// TIA Portal V19 export
FUNCTION "INPUT MAPING" : Void   // FC1, LAD
{ S7_Optimized_Access := 'TRUE' }
// stored: SetENOAutomatically false
BEGIN

REGION Network 1: "CPU RUN"
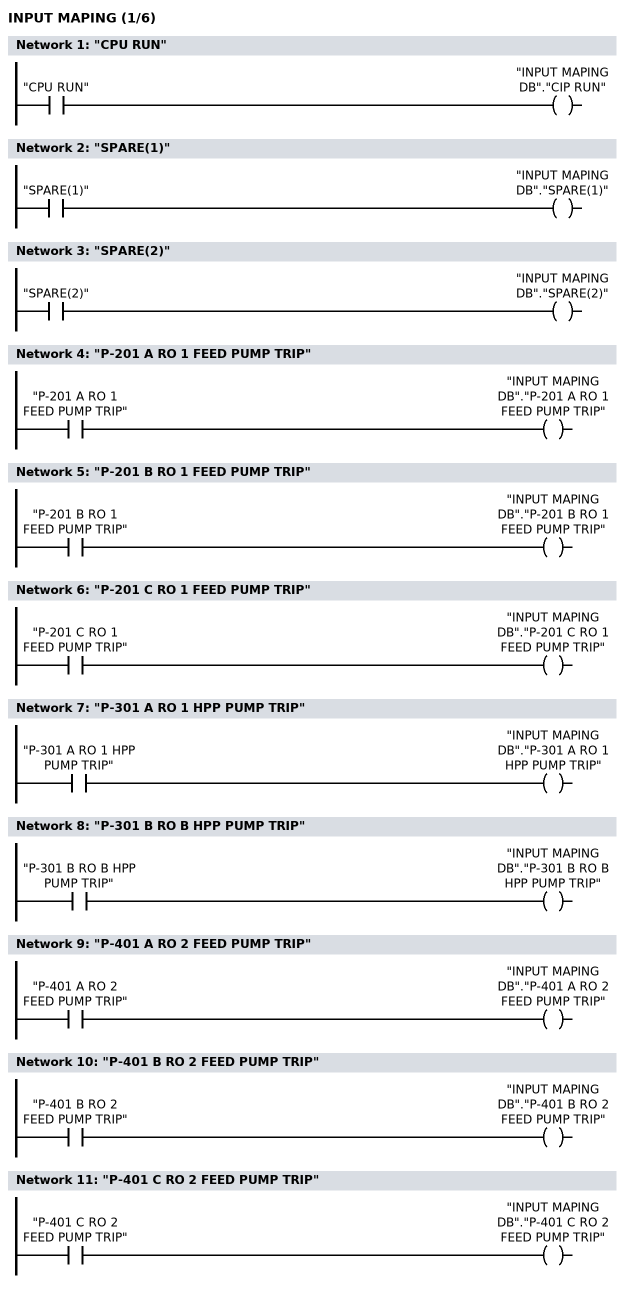
   RUNG wire#powerrail
      Contact( "CPU RUN" )
      Coil( "INPUT MAPING DB"."CIP RUN" )
   END_RUNG
   // the same network as SCL:
   "INPUT MAPING DB"."CIP RUN" := "CPU RUN";
END_REGION

REGION Network 2: "SPARE(1)"
   RUNG wire#powerrail
      Contact( "SPARE(1)" )
      Coil( "INPUT MAPING DB"."SPARE(1)" )
   END_RUNG
   // the same network as SCL:
   "INPUT MAPING DB"."SPARE(1)" := "SPARE(1)";
END_REGION

REGION Network 3: "SPARE(2)"
   RUNG wire#powerrail
      Contact( "SPARE(2)" )
      Coil( "INPUT MAPING DB"."SPARE(2)" )
   END_RUNG
   // the same network as SCL:
   "INPUT MAPING DB"."SPARE(2)" := "SPARE(2)";
END_REGION

REGION Network 4: "P-201 A RO 1 FEED PUMP TRIP"
   RUNG wire#powerrail
      Contact( "P-201 A RO 1 FEED PUMP TRIP" )
      Coil( "INPUT MAPING DB"."P-201 A RO 1 FEED PUMP TRIP" )
   END_RUNG
   // the same network as SCL:
   "INPUT MAPING DB"."P-201 A RO 1 FEED PUMP TRIP" := "P-201 A RO 1 FEED PUMP TRIP";
END_REGION

REGION Network 5: "P-201 B RO 1 FEED PUMP TRIP"
   RUNG wire#powerrail
      Contact( "P-201 B RO 1 FEED PUMP TRIP" )
      Coil( "INPUT MAPING DB"."P-201 B RO 1 FEED PUMP TRIP" )
   END_RUNG
   // the same network as SCL:
   "INPUT MAPING DB"."P-201 B RO 1 FEED PUMP TRIP" := "P-201 B RO 1 FEED PUMP TRIP";
END_REGION

REGION Network 6: "P-201 C RO 1 FEED PUMP TRIP"
   RUNG wire#powerrail
      Contact( "P-201 C RO 1 FEED PUMP TRIP" )
      Coil( "INPUT MAPING DB"."P-201 C RO 1 FEED PUMP TRIP" )
   END_RUNG
   // the same network as SCL:
   "INPUT MAPING DB"."P-201 C RO 1 FEED PUMP TRIP" := "P-201 C RO 1 FEED PUMP TRIP";
END_REGION

REGION Network 7: "P-301 A RO 1 HPP PUMP TRIP"
   RUNG wire#powerrail
      Contact( "P-301 A RO 1 HPP PUMP TRIP" )
      Coil( "INPUT MAPING DB"."P-301 A RO 1 HPP PUMP TRIP" )
   END_RUNG
   // the same network as SCL:
   "INPUT MAPING DB"."P-301 A RO 1 HPP PUMP TRIP" := "P-301 A RO 1 HPP PUMP TRIP";
END_REGION

REGION Network 8: "P-301 B RO B HPP PUMP TRIP"
   RUNG wire#powerrail
      Contact( "P-301 B RO B HPP PUMP TRIP" )
      Coil( "INPUT MAPING DB"."P-301 B RO B HPP PUMP TRIP" )
   END_RUNG
   // the same network as SCL:
   "INPUT MAPING DB"."P-301 B RO B HPP PUMP TRIP" := "P-301 B RO B HPP PUMP TRIP";
END_REGION

REGION Network 9: "P-401 A RO 2 FEED PUMP TRIP"
   RUNG wire#powerrail
      Contact( "P-401 A RO 2 FEED PUMP TRIP" )
      Coil( "INPUT MAPING DB"."P-401 A RO 2 FEED PUMP TRIP" )
   END_RUNG
   // the same network as SCL:
   "INPUT MAPING DB"."P-401 A RO 2 FEED PUMP TRIP" := "P-401 A RO 2 FEED PUMP TRIP";
END_REGION

REGION Network 10: "P-401 B RO 2 FEED PUMP TRIP"
   RUNG wire#powerrail
      Contact( "P-401 B RO 2 FEED PUMP TRIP" )
      Coil( "INPUT MAPING DB"."P-401 B RO 2 FEED PUMP TRIP" )
   END_RUNG
   // the same network as SCL:
   "INPUT MAPING DB"."P-401 B RO 2 FEED PUMP TRIP" := "P-401 B RO 2 FEED PUMP TRIP";
END_REGION

REGION Network 11: "P-401 C RO 2 FEED PUMP TRIP"
   RUNG wire#powerrail
      Contact( "P-401 C RO 2 FEED PUMP TRIP" )
      Coil( "INPUT MAPING DB"."P-401 C RO 2 FEED PUMP TRIP" )
   END_RUNG
   // the same network as SCL:
   "INPUT MAPING DB"."P-401 C RO 2 FEED PUMP TRIP" := "P-401 C RO 2 FEED PUMP TRIP";
END_REGION

REGION Network 12: "P 401 A RO 2 HPP PUMP TRIP"
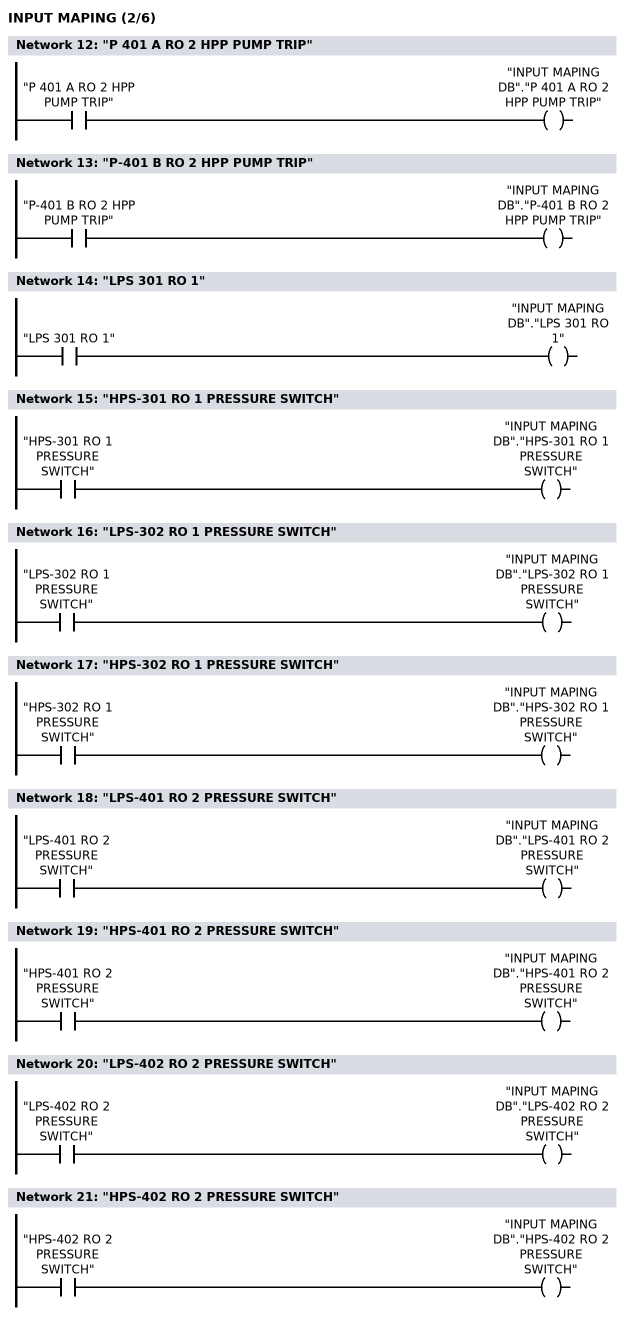
   RUNG wire#powerrail
      Contact( "P 401 A RO 2 HPP PUMP TRIP" )
      Coil( "INPUT MAPING DB"."P 401 A RO 2 HPP PUMP TRIP" )
   END_RUNG
   // the same network as SCL:
   "INPUT MAPING DB"."P 401 A RO 2 HPP PUMP TRIP" := "P 401 A RO 2 HPP PUMP TRIP";
END_REGION

REGION Network 13: "P-401 B RO 2 HPP PUMP TRIP"
   RUNG wire#powerrail
      Contact( "P-401 B RO 2 HPP PUMP TRIP" )
      Coil( "INPUT MAPING DB"."P-401 B RO 2 HPP PUMP TRIP" )
   END_RUNG
   // the same network as SCL:
   "INPUT MAPING DB"."P-401 B RO 2 HPP PUMP TRIP" := "P-401 B RO 2 HPP PUMP TRIP";
END_REGION

REGION Network 14: "LPS 301 RO 1"
   RUNG wire#powerrail
      Contact( "LPS 301 RO 1" )
      Coil( "INPUT MAPING DB"."LPS 301 RO 1" )
   END_RUNG
   // the same network as SCL:
   "INPUT MAPING DB"."LPS 301 RO 1" := "LPS 301 RO 1";
END_REGION

REGION Network 15: "HPS-301 RO 1 PRESSURE SWITCH"
   RUNG wire#powerrail
      Contact( "HPS-301 RO 1 PRESSURE SWITCH" )
      Coil( "INPUT MAPING DB"."HPS-301 RO 1 PRESSURE SWITCH" )
   END_RUNG
   // the same network as SCL:
   "INPUT MAPING DB"."HPS-301 RO 1 PRESSURE SWITCH" := "HPS-301 RO 1 PRESSURE SWITCH";
END_REGION

REGION Network 16: "LPS-302 RO 1 PRESSURE SWITCH"
   RUNG wire#powerrail
      Contact( "LPS-302 RO 1 PRESSURE SWITCH" )
      Coil( "INPUT MAPING DB"."LPS-302 RO 1 PRESSURE SWITCH" )
   END_RUNG
   // the same network as SCL:
   "INPUT MAPING DB"."LPS-302 RO 1 PRESSURE SWITCH" := "LPS-302 RO 1 PRESSURE SWITCH";
END_REGION

REGION Network 17: "HPS-302 RO 1 PRESSURE SWITCH"
   RUNG wire#powerrail
      Contact( "HPS-302 RO 1 PRESSURE SWITCH" )
      Coil( "INPUT MAPING DB"."HPS-302 RO 1 PRESSURE SWITCH" )
   END_RUNG
   // the same network as SCL:
   "INPUT MAPING DB"."HPS-302 RO 1 PRESSURE SWITCH" := "HPS-302 RO 1 PRESSURE SWITCH";
END_REGION

REGION Network 18: "LPS-401 RO 2 PRESSURE SWITCH"
   RUNG wire#powerrail
      Contact( "LPS-401 RO 2 PRESSURE SWITCH" )
      Coil( "INPUT MAPING DB"."LPS-401 RO 2 PRESSURE SWITCH" )
   END_RUNG
   // the same network as SCL:
   "INPUT MAPING DB"."LPS-401 RO 2 PRESSURE SWITCH" := "LPS-401 RO 2 PRESSURE SWITCH";
END_REGION

REGION Network 19: "HPS-401 RO 2 PRESSURE SWITCH"
   RUNG wire#powerrail
      Contact( "HPS-401 RO 2 PRESSURE SWITCH" )
      Coil( "INPUT MAPING DB"."HPS-401 RO 2 PRESSURE SWITCH" )
   END_RUNG
   // the same network as SCL:
   "INPUT MAPING DB"."HPS-401 RO 2 PRESSURE SWITCH" := "HPS-401 RO 2 PRESSURE SWITCH";
END_REGION

REGION Network 20: "LPS-402 RO 2 PRESSURE SWITCH"
   RUNG wire#powerrail
      Contact( "LPS-402 RO 2 PRESSURE SWITCH" )
      Coil( "INPUT MAPING DB"."LPS-402 RO 2 PRESSURE SWITCH" )
   END_RUNG
   // the same network as SCL:
   "INPUT MAPING DB"."LPS-402 RO 2 PRESSURE SWITCH" := "LPS-402 RO 2 PRESSURE SWITCH";
END_REGION

REGION Network 21: "HPS-402 RO 2 PRESSURE SWITCH"
   RUNG wire#powerrail
      Contact( "HPS-402 RO 2 PRESSURE SWITCH" )
      Coil( "INPUT MAPING DB"."HPS-402 RO 2 PRESSURE SWITCH" )
   END_RUNG
   // the same network as SCL:
   "INPUT MAPING DB"."HPS-402 RO 2 PRESSURE SWITCH" := "HPS-402 RO 2 PRESSURE SWITCH";
END_REGION

REGION Network 22: "DP-703 RO 1 DOSER LEVEL SWITCH"
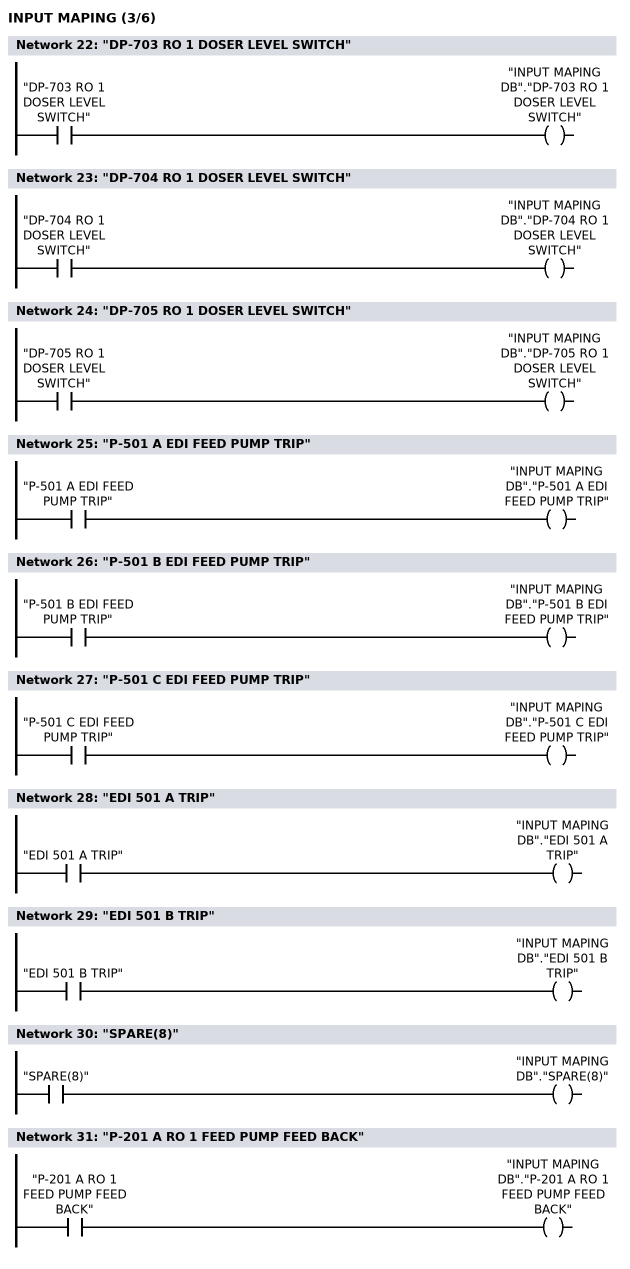
   RUNG wire#powerrail
      Contact( "DP-703 RO 1 DOSER LEVEL SWITCH" )
      Coil( "INPUT MAPING DB"."DP-703 RO 1 DOSER LEVEL SWITCH" )
   END_RUNG
   // the same network as SCL:
   "INPUT MAPING DB"."DP-703 RO 1 DOSER LEVEL SWITCH" := "DP-703 RO 1 DOSER LEVEL SWITCH";
END_REGION

REGION Network 23: "DP-704 RO 1 DOSER LEVEL SWITCH"
   RUNG wire#powerrail
      Contact( "DP-704 RO 1 DOSER LEVEL SWITCH" )
      Coil( "INPUT MAPING DB"."DP-704 RO 1 DOSER LEVEL SWITCH" )
   END_RUNG
   // the same network as SCL:
   "INPUT MAPING DB"."DP-704 RO 1 DOSER LEVEL SWITCH" := "DP-704 RO 1 DOSER LEVEL SWITCH";
END_REGION

REGION Network 24: "DP-705 RO 1 DOSER LEVEL SWITCH"
   RUNG wire#powerrail
      Contact( "DP-705 RO 1 DOSER LEVEL SWITCH" )
      Coil( "INPUT MAPING DB"."DP-705 RO 1 DOSER LEVEL SWITCH" )
   END_RUNG
   // the same network as SCL:
   "INPUT MAPING DB"."DP-705 RO 1 DOSER LEVEL SWITCH" := "DP-705 RO 1 DOSER LEVEL SWITCH";
END_REGION

REGION Network 25: "P-501 A EDI FEED PUMP TRIP"
   RUNG wire#powerrail
      Contact( "P-501 A EDI FEED PUMP TRIP" )
      Coil( "INPUT MAPING DB"."P-501 A EDI FEED PUMP TRIP" )
   END_RUNG
   // the same network as SCL:
   "INPUT MAPING DB"."P-501 A EDI FEED PUMP TRIP" := "P-501 A EDI FEED PUMP TRIP";
END_REGION

REGION Network 26: "P-501 B EDI FEED PUMP TRIP"
   RUNG wire#powerrail
      Contact( "P-501 B EDI FEED PUMP TRIP" )
      Coil( "INPUT MAPING DB"."P-501 B EDI FEED PUMP TRIP" )
   END_RUNG
   // the same network as SCL:
   "INPUT MAPING DB"."P-501 B EDI FEED PUMP TRIP" := "P-501 B EDI FEED PUMP TRIP";
END_REGION

REGION Network 27: "P-501 C EDI FEED PUMP TRIP"
   RUNG wire#powerrail
      Contact( "P-501 C EDI FEED PUMP TRIP" )
      Coil( "INPUT MAPING DB"."P-501 C EDI FEED PUMP TRIP" )
   END_RUNG
   // the same network as SCL:
   "INPUT MAPING DB"."P-501 C EDI FEED PUMP TRIP" := "P-501 C EDI FEED PUMP TRIP";
END_REGION

REGION Network 28: "EDI 501 A TRIP"
   RUNG wire#powerrail
      Contact( "EDI 501 A TRIP" )
      Coil( "INPUT MAPING DB"."EDI 501 A TRIP" )
   END_RUNG
   // the same network as SCL:
   "INPUT MAPING DB"."EDI 501 A TRIP" := "EDI 501 A TRIP";
END_REGION

REGION Network 29: "EDI 501 B TRIP"
   RUNG wire#powerrail
      Contact( "EDI 501 B TRIP" )
      Coil( "INPUT MAPING DB"."EDI 501 B TRIP" )
   END_RUNG
   // the same network as SCL:
   "INPUT MAPING DB"."EDI 501 B TRIP" := "EDI 501 B TRIP";
END_REGION

REGION Network 30: "SPARE(8)"
   RUNG wire#powerrail
      Contact( "SPARE(8)" )
      Coil( "INPUT MAPING DB"."SPARE(8)" )
   END_RUNG
   // the same network as SCL:
   "INPUT MAPING DB"."SPARE(8)" := "SPARE(8)";
END_REGION

REGION Network 31: "P-201 A RO 1 FEED PUMP FEED BACK"
   RUNG wire#powerrail
      Contact( "P-201 A RO 1 FEED PUMP FEED BACK" )
      Coil( "INPUT MAPING DB"."P-201 A RO 1 FEED PUMP FEED BACK" )
   END_RUNG
   // the same network as SCL:
   "INPUT MAPING DB"."P-201 A RO 1 FEED PUMP FEED BACK" := "P-201 A RO 1 FEED PUMP FEED BACK";
END_REGION

REGION Network 32: "P-201 B RO 1 FEED PUMP FEED BACK"
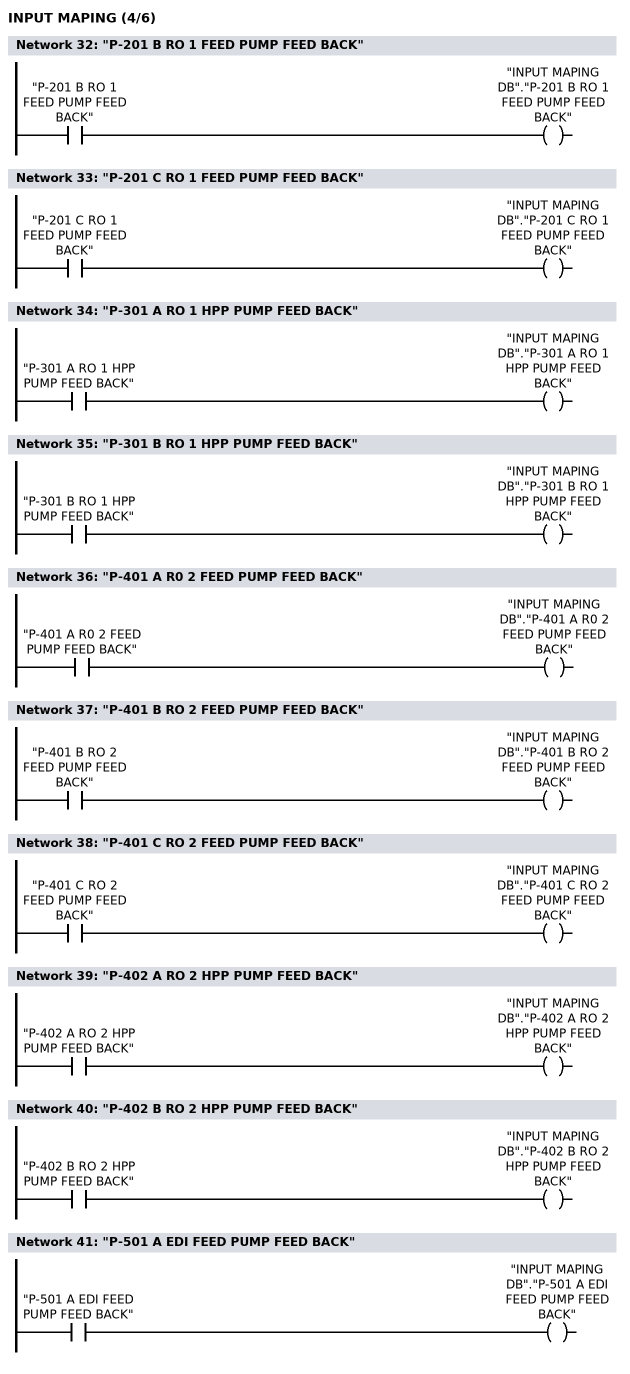
   RUNG wire#powerrail
      Contact( "P-201 B RO 1 FEED PUMP FEED BACK" )
      Coil( "INPUT MAPING DB"."P-201 B RO 1 FEED PUMP FEED BACK" )
   END_RUNG
   // the same network as SCL:
   "INPUT MAPING DB"."P-201 B RO 1 FEED PUMP FEED BACK" := "P-201 B RO 1 FEED PUMP FEED BACK";
END_REGION

REGION Network 33: "P-201 C RO 1 FEED PUMP FEED BACK"
   RUNG wire#powerrail
      Contact( "P-201 C RO 1 FEED PUMP FEED BACK" )
      Coil( "INPUT MAPING DB"."P-201 C RO 1 FEED PUMP FEED BACK" )
   END_RUNG
   // the same network as SCL:
   "INPUT MAPING DB"."P-201 C RO 1 FEED PUMP FEED BACK" := "P-201 C RO 1 FEED PUMP FEED BACK";
END_REGION

REGION Network 34: "P-301 A RO 1 HPP PUMP FEED BACK"
   RUNG wire#powerrail
      Contact( "P-301 A RO 1 HPP PUMP FEED BACK" )
      Coil( "INPUT MAPING DB"."P-301 A RO 1 HPP PUMP FEED BACK" )
   END_RUNG
   // the same network as SCL:
   "INPUT MAPING DB"."P-301 A RO 1 HPP PUMP FEED BACK" := "P-301 A RO 1 HPP PUMP FEED BACK";
END_REGION

REGION Network 35: "P-301 B RO 1 HPP PUMP FEED BACK"
   RUNG wire#powerrail
      Contact( "P-301 B RO 1 HPP PUMP FEED BACK" )
      Coil( "INPUT MAPING DB"."P-301 B RO 1 HPP PUMP FEED BACK" )
   END_RUNG
   // the same network as SCL:
   "INPUT MAPING DB"."P-301 B RO 1 HPP PUMP FEED BACK" := "P-301 B RO 1 HPP PUMP FEED BACK";
END_REGION

REGION Network 36: "P-401 A R0 2 FEED PUMP FEED BACK"
   RUNG wire#powerrail
      Contact( "P-401 A R0 2 FEED PUMP FEED BACK" )
      Coil( "INPUT MAPING DB"."P-401 A R0 2 FEED PUMP FEED BACK" )
   END_RUNG
   // the same network as SCL:
   "INPUT MAPING DB"."P-401 A R0 2 FEED PUMP FEED BACK" := "P-401 A R0 2 FEED PUMP FEED BACK";
END_REGION

REGION Network 37: "P-401 B RO 2 FEED PUMP FEED BACK"
   RUNG wire#powerrail
      Contact( "P-401 B RO 2 FEED PUMP FEED BACK" )
      Coil( "INPUT MAPING DB"."P-401 B RO 2 FEED PUMP FEED BACK" )
   END_RUNG
   // the same network as SCL:
   "INPUT MAPING DB"."P-401 B RO 2 FEED PUMP FEED BACK" := "P-401 B RO 2 FEED PUMP FEED BACK";
END_REGION

REGION Network 38: "P-401 C RO 2 FEED PUMP FEED BACK"
   RUNG wire#powerrail
      Contact( "P-401 C RO 2 FEED PUMP FEED BACK" )
      Coil( "INPUT MAPING DB"."P-401 C RO 2 FEED PUMP FEED BACK" )
   END_RUNG
   // the same network as SCL:
   "INPUT MAPING DB"."P-401 C RO 2 FEED PUMP FEED BACK" := "P-401 C RO 2 FEED PUMP FEED BACK";
END_REGION

REGION Network 39: "P-402 A RO 2 HPP PUMP FEED BACK"
   RUNG wire#powerrail
      Contact( "P-402 A RO 2 HPP PUMP FEED BACK" )
      Coil( "INPUT MAPING DB"."P-402 A RO 2 HPP PUMP FEED BACK" )
   END_RUNG
   // the same network as SCL:
   "INPUT MAPING DB"."P-402 A RO 2 HPP PUMP FEED BACK" := "P-402 A RO 2 HPP PUMP FEED BACK";
END_REGION

REGION Network 40: "P-402 B RO 2 HPP PUMP FEED BACK"
   RUNG wire#powerrail
      Contact( "P-402 B RO 2 HPP PUMP FEED BACK" )
      Coil( "INPUT MAPING DB"."P-402 B RO 2 HPP PUMP FEED BACK" )
   END_RUNG
   // the same network as SCL:
   "INPUT MAPING DB"."P-402 B RO 2 HPP PUMP FEED BACK" := "P-402 B RO 2 HPP PUMP FEED BACK";
END_REGION

REGION Network 41: "P-501 A EDI FEED PUMP FEED BACK"
   RUNG wire#powerrail
      Contact( "P-501 A EDI FEED PUMP FEED BACK" )
      Coil( "INPUT MAPING DB"."P-501 A EDI FEED PUMP FEED BACK" )
   END_RUNG
   // the same network as SCL:
   "INPUT MAPING DB"."P-501 A EDI FEED PUMP FEED BACK" := "P-501 A EDI FEED PUMP FEED BACK";
END_REGION

REGION Network 42: "P-501 B EDI FEED PUMP FEED BACK"
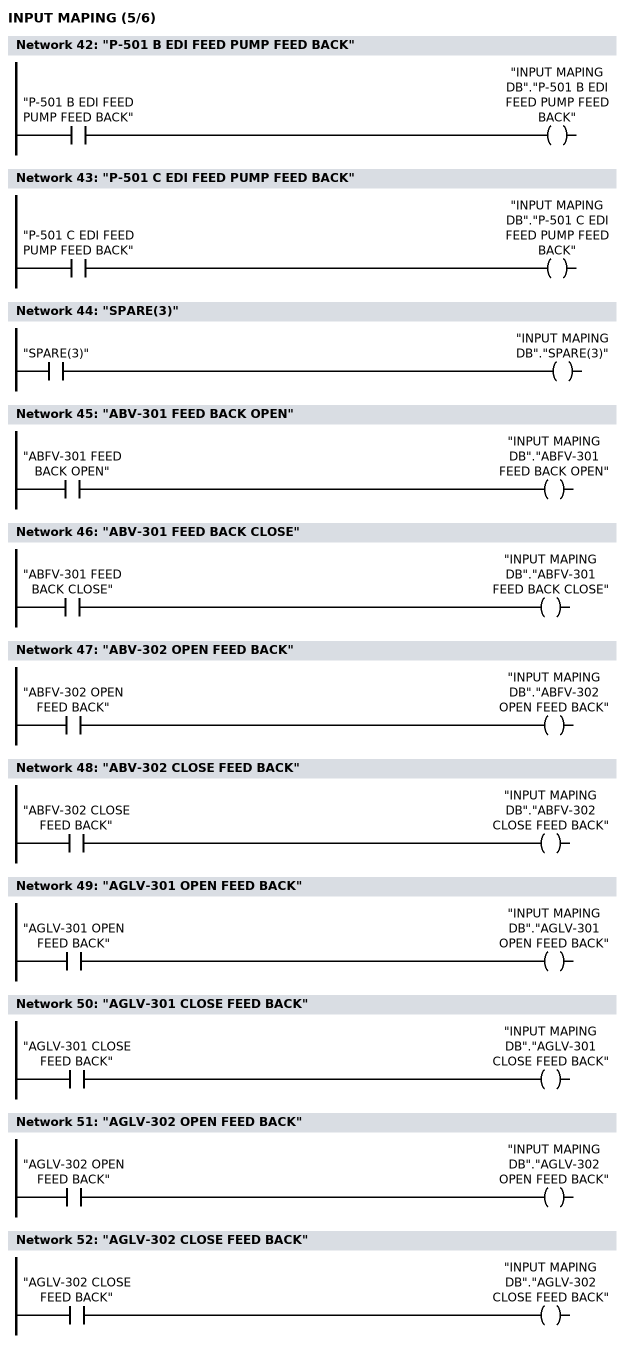
   RUNG wire#powerrail
      Contact( "P-501 B EDI FEED PUMP FEED BACK" )
      Coil( "INPUT MAPING DB"."P-501 B EDI FEED PUMP FEED BACK" )
   END_RUNG
   // the same network as SCL:
   "INPUT MAPING DB"."P-501 B EDI FEED PUMP FEED BACK" := "P-501 B EDI FEED PUMP FEED BACK";
END_REGION

REGION Network 43: "P-501 C EDI FEED PUMP FEED BACK"
   RUNG wire#powerrail
      Contact( "P-501 C EDI FEED PUMP FEED BACK" )
      Coil( "INPUT MAPING DB"."P-501 C EDI FEED PUMP FEED BACK" )
   END_RUNG
   // the same network as SCL:
   "INPUT MAPING DB"."P-501 C EDI FEED PUMP FEED BACK" := "P-501 C EDI FEED PUMP FEED BACK";
END_REGION

REGION Network 44: "SPARE(3)"
   RUNG wire#powerrail
      Contact( "SPARE(3)" )
      Coil( "INPUT MAPING DB"."SPARE(3)" )
   END_RUNG
   // the same network as SCL:
   "INPUT MAPING DB"."SPARE(3)" := "SPARE(3)";
END_REGION

REGION Network 45: "ABV-301 FEED BACK OPEN"
   RUNG wire#powerrail
      Contact( "ABFV-301 FEED BACK OPEN" )
      Coil( "INPUT MAPING DB"."ABFV-301 FEED BACK OPEN" )
   END_RUNG
   // the same network as SCL:
   "INPUT MAPING DB"."ABFV-301 FEED BACK OPEN" := "ABFV-301 FEED BACK OPEN";
END_REGION

REGION Network 46: "ABV-301 FEED BACK CLOSE"
   RUNG wire#powerrail
      Contact( "ABFV-301 FEED BACK CLOSE" )
      Coil( "INPUT MAPING DB"."ABFV-301 FEED BACK CLOSE" )
   END_RUNG
   // the same network as SCL:
   "INPUT MAPING DB"."ABFV-301 FEED BACK CLOSE" := "ABFV-301 FEED BACK CLOSE";
END_REGION

REGION Network 47: "ABV-302 OPEN FEED BACK"
   RUNG wire#powerrail
      Contact( "ABFV-302 OPEN FEED BACK" )
      Coil( "INPUT MAPING DB"."ABFV-302 OPEN FEED BACK" )
   END_RUNG
   // the same network as SCL:
   "INPUT MAPING DB"."ABFV-302 OPEN FEED BACK" := "ABFV-302 OPEN FEED BACK";
END_REGION

REGION Network 48: "ABV-302 CLOSE FEED BACK"
   RUNG wire#powerrail
      Contact( "ABFV-302 CLOSE FEED BACK" )
      Coil( "INPUT MAPING DB"."ABFV-302 CLOSE FEED BACK" )
   END_RUNG
   // the same network as SCL:
   "INPUT MAPING DB"."ABFV-302 CLOSE FEED BACK" := "ABFV-302 CLOSE FEED BACK";
END_REGION

REGION Network 49: "AGLV-301 OPEN FEED BACK"
   RUNG wire#powerrail
      Contact( "AGLV-301 OPEN FEED BACK" )
      Coil( "INPUT MAPING DB"."AGLV-301 OPEN FEED BACK" )
   END_RUNG
   // the same network as SCL:
   "INPUT MAPING DB"."AGLV-301 OPEN FEED BACK" := "AGLV-301 OPEN FEED BACK";
END_REGION

REGION Network 50: "AGLV-301 CLOSE FEED BACK"
   RUNG wire#powerrail
      Contact( "AGLV-301 CLOSE FEED BACK" )
      Coil( "INPUT MAPING DB"."AGLV-301 CLOSE FEED BACK" )
   END_RUNG
   // the same network as SCL:
   "INPUT MAPING DB"."AGLV-301 CLOSE FEED BACK" := "AGLV-301 CLOSE FEED BACK";
END_REGION

REGION Network 51: "AGLV-302 OPEN FEED BACK"
   RUNG wire#powerrail
      Contact( "AGLV-302 OPEN FEED BACK" )
      Coil( "INPUT MAPING DB"."AGLV-302 OPEN FEED BACK" )
   END_RUNG
   // the same network as SCL:
   "INPUT MAPING DB"."AGLV-302 OPEN FEED BACK" := "AGLV-302 OPEN FEED BACK";
END_REGION

REGION Network 52: "AGLV-302 CLOSE FEED BACK"
   RUNG wire#powerrail
      Contact( "AGLV-302 CLOSE FEED BACK" )
      Coil( "INPUT MAPING DB"."AGLV-302 CLOSE FEED BACK" )
   END_RUNG
   // the same network as SCL:
   "INPUT MAPING DB"."AGLV-302 CLOSE FEED BACK" := "AGLV-302 CLOSE FEED BACK";
END_REGION

REGION Network 53: "AGLV-401 OPEN FEED BACK"
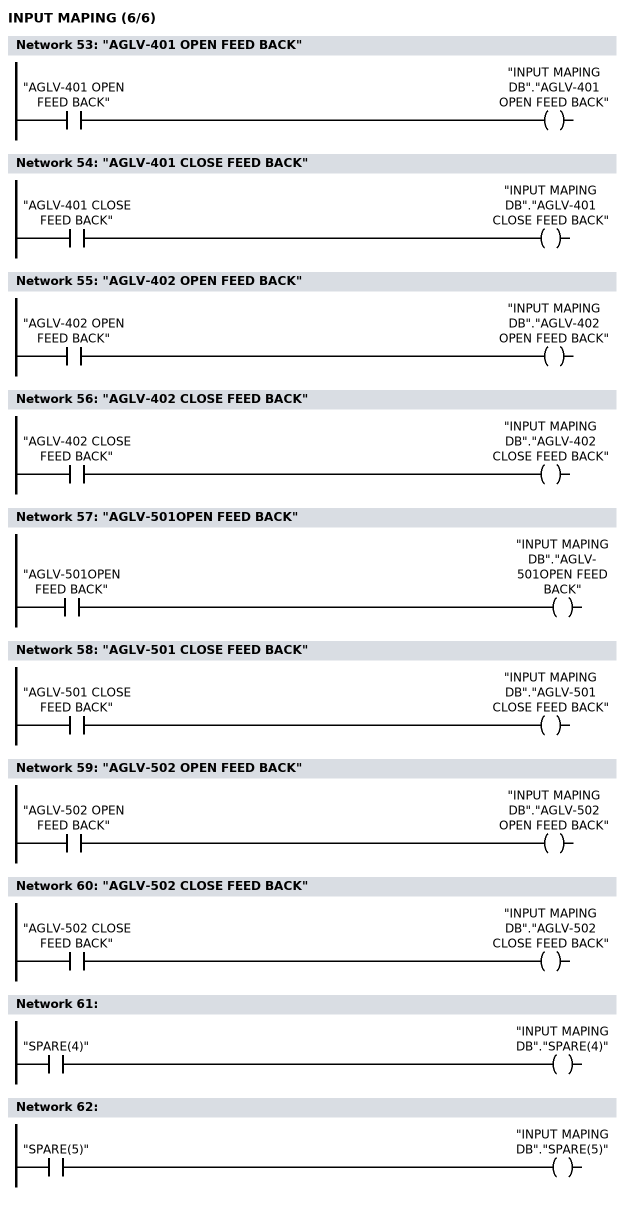
   RUNG wire#powerrail
      Contact( "AGLV-401 OPEN FEED BACK" )
      Coil( "INPUT MAPING DB"."AGLV-401 OPEN FEED BACK" )
   END_RUNG
   // the same network as SCL:
   "INPUT MAPING DB"."AGLV-401 OPEN FEED BACK" := "AGLV-401 OPEN FEED BACK";
END_REGION

REGION Network 54: "AGLV-401 CLOSE FEED BACK"
   RUNG wire#powerrail
      Contact( "AGLV-401 CLOSE FEED BACK" )
      Coil( "INPUT MAPING DB"."AGLV-401 CLOSE FEED BACK" )
   END_RUNG
   // the same network as SCL:
   "INPUT MAPING DB"."AGLV-401 CLOSE FEED BACK" := "AGLV-401 CLOSE FEED BACK";
END_REGION

REGION Network 55: "AGLV-402 OPEN FEED BACK"
   RUNG wire#powerrail
      Contact( "AGLV-402 OPEN FEED BACK" )
      Coil( "INPUT MAPING DB"."AGLV-402 OPEN FEED BACK" )
   END_RUNG
   // the same network as SCL:
   "INPUT MAPING DB"."AGLV-402 OPEN FEED BACK" := "AGLV-402 OPEN FEED BACK";
END_REGION

REGION Network 56: "AGLV-402 CLOSE FEED BACK"
   RUNG wire#powerrail
      Contact( "AGLV-402 CLOSE FEED BACK" )
      Coil( "INPUT MAPING DB"."AGLV-402 CLOSE FEED BACK" )
   END_RUNG
   // the same network as SCL:
   "INPUT MAPING DB"."AGLV-402 CLOSE FEED BACK" := "AGLV-402 CLOSE FEED BACK";
END_REGION

REGION Network 57: "AGLV-501OPEN FEED BACK"
   RUNG wire#powerrail
      Contact( "AGLV-501OPEN FEED BACK" )
      Coil( "INPUT MAPING DB"."AGLV-501OPEN FEED BACK" )
   END_RUNG
   // the same network as SCL:
   "INPUT MAPING DB"."AGLV-501OPEN FEED BACK" := "AGLV-501OPEN FEED BACK";
END_REGION

REGION Network 58: "AGLV-501 CLOSE FEED BACK"
   RUNG wire#powerrail
      Contact( "AGLV-501 CLOSE FEED BACK" )
      Coil( "INPUT MAPING DB"."AGLV-501 CLOSE FEED BACK" )
   END_RUNG
   // the same network as SCL:
   "INPUT MAPING DB"."AGLV-501 CLOSE FEED BACK" := "AGLV-501 CLOSE FEED BACK";
END_REGION

REGION Network 59: "AGLV-502 OPEN FEED BACK"
   RUNG wire#powerrail
      Contact( "AGLV-502 OPEN FEED BACK" )
      Coil( "INPUT MAPING DB"."AGLV-502 OPEN FEED BACK" )
   END_RUNG
   // the same network as SCL:
   "INPUT MAPING DB"."AGLV-502 OPEN FEED BACK" := "AGLV-502 OPEN FEED BACK";
END_REGION

REGION Network 60: "AGLV-502 CLOSE FEED BACK"
   RUNG wire#powerrail
      Contact( "AGLV-502 CLOSE FEED BACK" )
      Coil( "INPUT MAPING DB"."AGLV-502 CLOSE FEED BACK" )
   END_RUNG
   // the same network as SCL:
   "INPUT MAPING DB"."AGLV-502 CLOSE FEED BACK" := "AGLV-502 CLOSE FEED BACK";
END_REGION

REGION Network 61
   RUNG wire#powerrail
      Contact( "SPARE(4)" )
      Coil( "INPUT MAPING DB"."SPARE(4)" )
   END_RUNG
   // the same network as SCL:
   "INPUT MAPING DB"."SPARE(4)" := "SPARE(4)";
END_REGION

REGION Network 62
   RUNG wire#powerrail
      Contact( "SPARE(5)" )
      Coil( "INPUT MAPING DB"."SPARE(5)" )
   END_RUNG
   // the same network as SCL:
   "INPUT MAPING DB"."SPARE(5)" := "SPARE(5)";
END_REGION
END_FUNCTION
